(* Schneider Machine Expert - Basic project Tarea1C3_TomasMoreno, file version 2.7.0.0 *)
(* ProjectInformations: Name=Nuevo proyecto *)

HARDWARE
  Cpu 0: TM221CE16R
  EthernetConfiguration: NetworkName=M221, IpAllocationMode=FixedAddress, IpAddress=0.0.0.0, SubnetMask=0.0.0.0
  SerialLineConfiguration: Baud=Baud19200, Parity=ParityEven, DataBits=DataBits8, StopBits=StopBits1, PhysicalMedium=PhysicalMediumRs485, TransmissionMode=TransmissionModeModbusRtu, SlaveId=1, Addressing=SlaveAddressing
  MastTask: UsePeriodScanMode=false, PeriodScan=100
  FastTask: Period=255
  CpuBehavior: StartingMode=StartAsPreviousState, AutoSaveRamOnEeprom=true, WatchdogPeriod=250

SYMBOLS  (address, symbol, comment, settings)
  %M0         "PARTIR"
  %M1         "PARAR"
  %M2         "AUTOMATICO"
  %M3         "MANUAL"
  %M4         "RESETEO"
  %M5         "PARADA DE EMERGENCIA"
  %M6         "SENSOR TRANSPORTE"
  %M7         "SENSOR CONTADOR CP"
  %M8         "SENSOR CONTADOR CG"
  %M9         "IMPULSADOR CAJAS (MANUAL)"
  %M20        "LED PARTIR"
  %M21        "LED RESET"
  %M22        "LED PARAR"
  %M23        "LED FUNCIONAMIENTO SISTEMA"
  %M24        "LED CONTADOR CP"
  %M25        "LED CONTADOR CG"
  %M26        "CORREA PRINCIPAL"
  %M27        "TRANSPORTE ADELANTE"
  %M28        "TRANSPORTE CG"
  %M29        "TRANSPORTE CP"
  %M30        "CORREA CAJAS GRANDES"
  %M31        "CORREA CAJAS PEQUEÑAS"
  %M32        "EMISOR DE CAJAS"
  %M33        "LED IMPULSADOR MANUAL"
  %M50        "ARRANQUE SISTEMA"
  %M61        "S_TRANSP_CG"
  %M62        "S_TRANSP_CP"
  %M63        "H_TRANSP_CG"
  %M64        "H_TRANSP_CP"
  %S6       SB_TB1S  "Base de tiempo de 1 s generada por un reloj interno"
  %TM0        [Type=TOF, Preset=1, Base=OneSecond]
  %TM1        [Type=TOF, Preset=1, Base=OneSecond]
  %C0         [Preset=1]
  %C1         [Preset=1]

POU Nuevo POU
  (* SectionNumber=1 *)

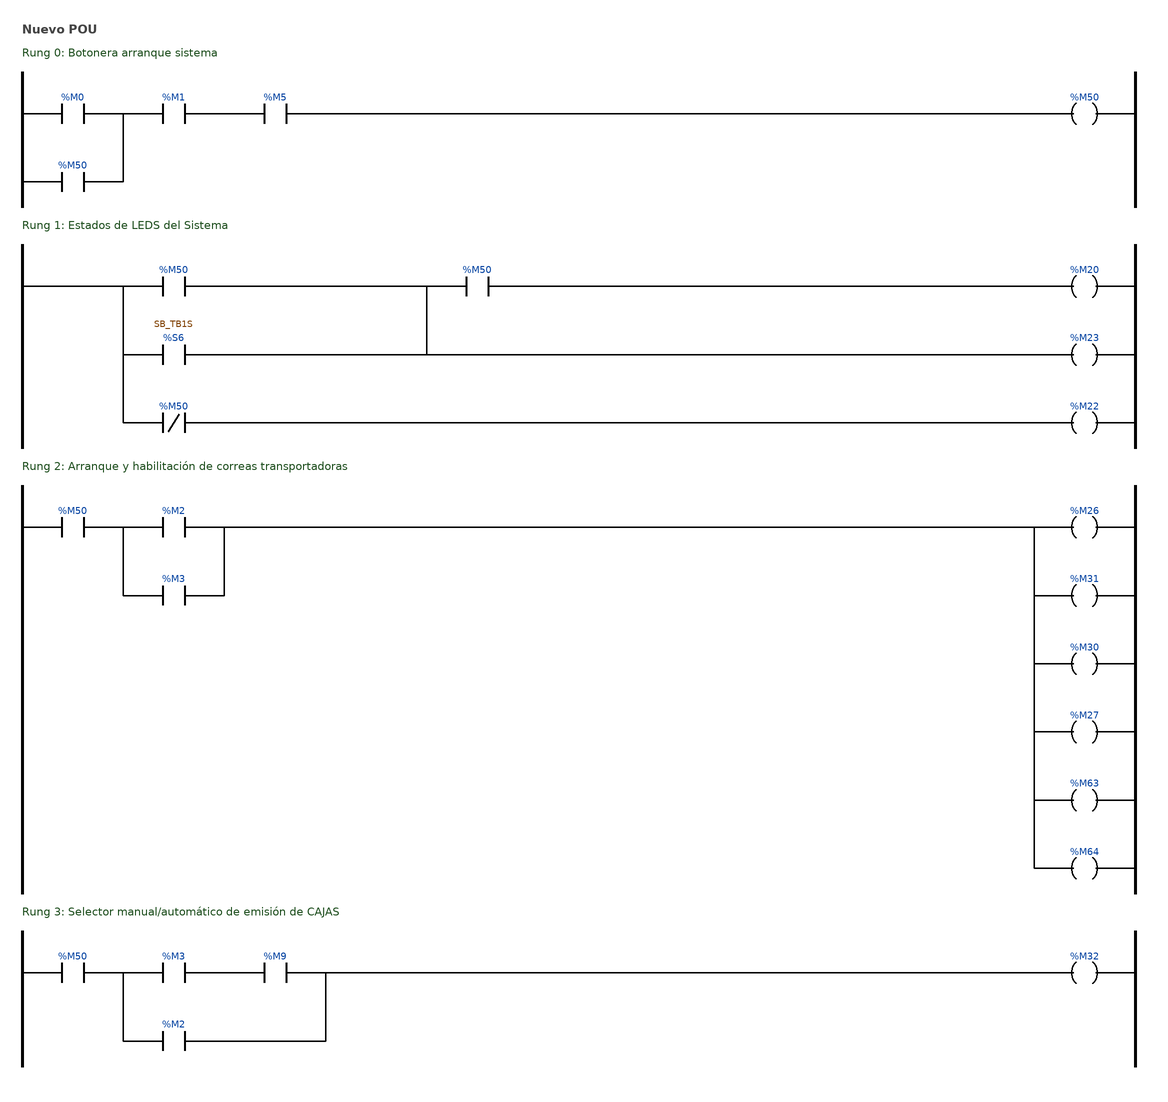

// Rung 0: Botonera arranque sistema
  LD %M0
  OR %M50
  AND %M1
  AND %M5
  ST %M50
  // as ST:
  //   %M50 := (%M0 OR %M50) AND %M1 AND %M5;

// Rung 1: Estados de LEDS del Sistema
  LD 1
  MPS
  AND( %M50
  OR %S6                  (* SB_TB1S *)
  )
  MPS
  AND %M50
  ST %M20
  MPP
  ST %M23
  MPP
  ANDN %M50
  ST %M22
  // as ST:
  //   %M20 := (%M50 OR SB_TB1S) AND %M50;
  //   %M23 := %M50 OR SB_TB1S;
  //   %M22 := NOT %M50;

// Rung 2: Arranque y habilitación de correas transportadoras
  LD %M50
  AND( %M2
  OR %M3
  )
  ST %M26
  ST %M31
  ST %M30
  ST %M27
  ST %M63
  ST %M64
  // as ST:
  //   %M26 := %M50 AND (%M2 OR %M3);
  //   %M31 := %M50 AND (%M2 OR %M3);
  //   %M30 := %M50 AND (%M2 OR %M3);
  //   %M27 := %M50 AND (%M2 OR %M3);
  //   %M63 := %M50 AND (%M2 OR %M3);
  //   %M64 := %M50 AND (%M2 OR %M3);

// Rung 3: Selector manual/automático de emisión de CAJAS
  LD %M50
  AND( %M3
  AND %M9
  OR %M2
  )
  ST %M32
  // as ST:
  //   %M32 := %M50 AND (%M3 AND %M9 OR %M2);

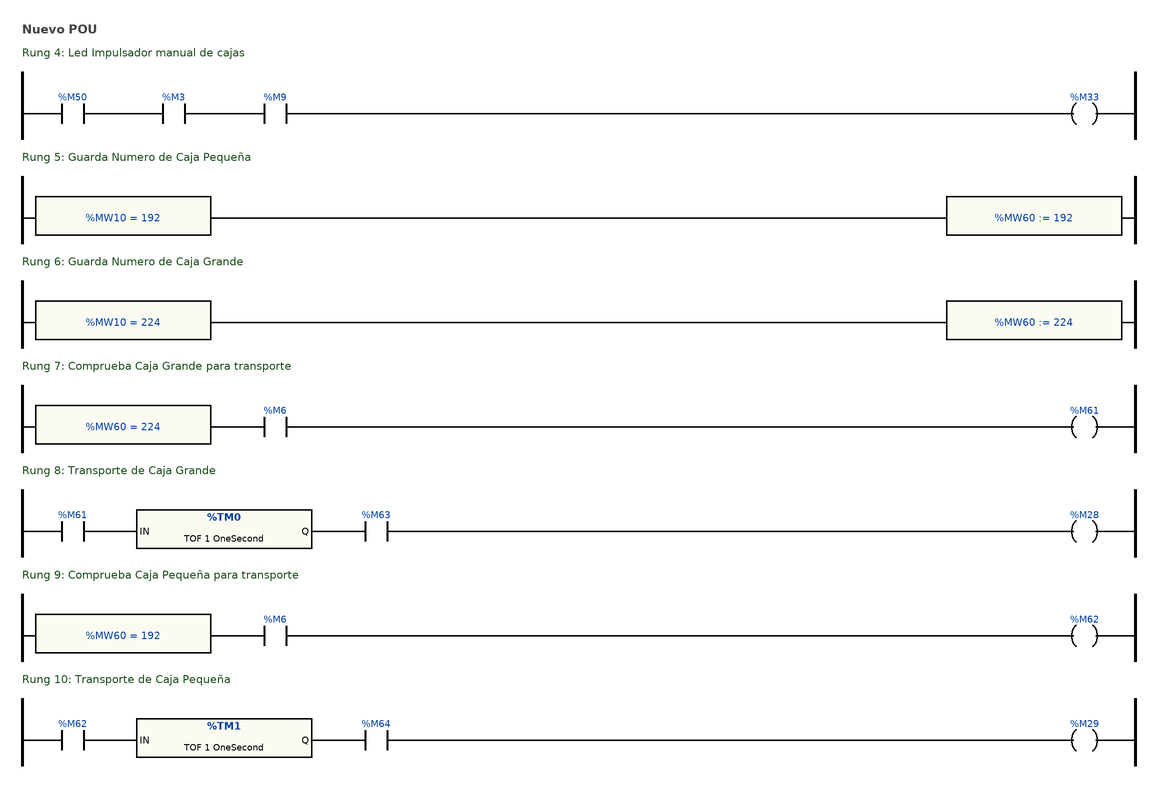

// Rung 4: Led Impulsador manual de cajas
  LD %M50
  AND %M3
  AND %M9
  ST %M33
  // as ST:
  //   %M33 := %M50 AND %M3 AND %M9;

// Rung 5: Guarda Numero de Caja Pequeña
  LD [ %MW10 = 192 ]
  [ %MW60 := 192 ]
  // as ST:
  //   IF %MW10 = 192 THEN %MW60 := 192; END_IF;

// Rung 6: Guarda Numero de Caja Grande
  LD [ %MW10 = 224 ]
  [ %MW60 := 224 ]
  // as ST:
  //   IF %MW10 = 224 THEN %MW60 := 224; END_IF;

// Rung 7: Comprueba Caja Grande para transporte
  LD [ %MW60 = 224 ]
  AND %M6
  ST %M61
  // as ST:
  //   %M61 := %MW60 = 224 AND %M6;

// Rung 8: Transporte de Caja Grande
  BLK %TM0
  LD %M61
  IN
  OUT_BLK
  LD Q
  AND %M63
  ST %M28
  END_BLK
  // as ST:
  //   %TM0(IN := %M61);
  //   %M28 := %TM0.Q AND %M63;

// Rung 9: Comprueba Caja Pequeña para transporte
  LD [ %MW60 = 192 ]
  AND %M6
  ST %M62
  // as ST:
  //   %M62 := %MW60 = 192 AND %M6;

// Rung 10: Transporte de Caja Pequeña
  BLK %TM1
  LD %M62
  IN
  OUT_BLK
  LD Q
  AND %M64
  ST %M29
  END_BLK
  // as ST:
  //   %TM1(IN := %M62);
  //   %M29 := %TM1.Q AND %M64;

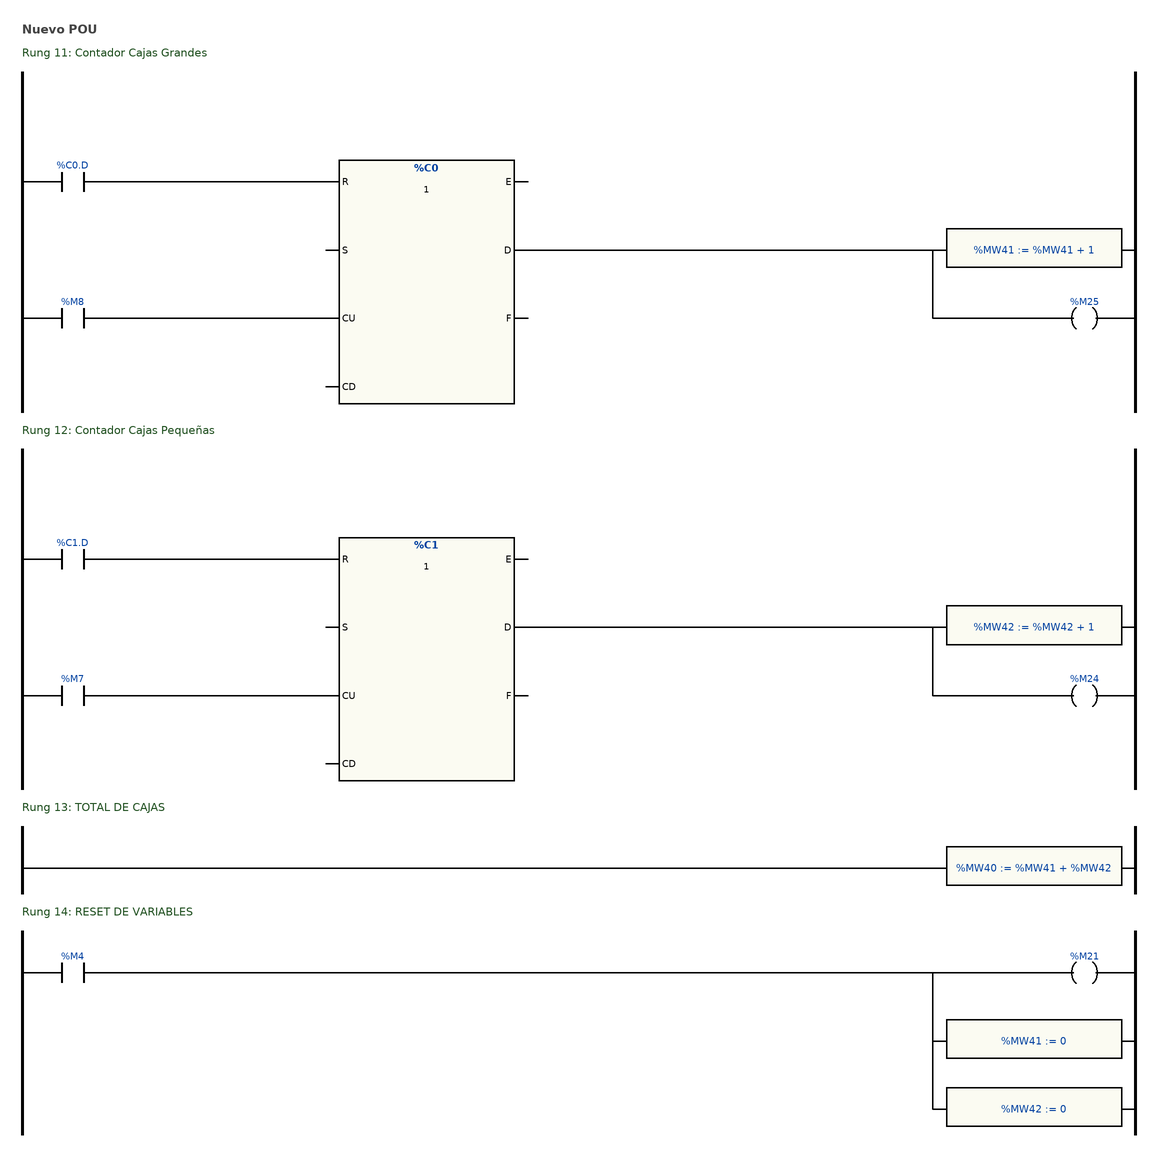

// Rung 11: Contador Cajas Grandes
  BLK %C0
  LD %C0.D
  R
  LD %M8
  CU
  OUT_BLK
  LD D
  [ %MW41 := %MW41 + 1 ]
  ST %M25
  END_BLK
  // as ST:
  //   %C0(R := %C0.D, CU := %M8);
  //   IF %C0.D THEN %MW41 := %MW41 + 1; END_IF;
  //   %M25 := %C0.D;

// Rung 12: Contador Cajas Pequeñas
  BLK %C1
  LD %C1.D
  R
  LD %M7
  CU
  OUT_BLK
  LD D
  [ %MW42 := %MW42 + 1 ]
  ST %M24
  END_BLK
  // as ST:
  //   %C1(R := %C1.D, CU := %M7);
  //   IF %C1.D THEN %MW42 := %MW42 + 1; END_IF;
  //   %M24 := %C1.D;

// Rung 13: TOTAL DE CAJAS
  LD 1
  [ %MW40 := %MW41 + %MW42 ]
  // as ST:
  //   %MW40 := %MW41 + %MW42;

// Rung 14: RESET DE VARIABLES
  LD %M4
  ST %M21
  [ %MW41 := 0 ]
  [ %MW42 := 0 ]
  // as ST:
  //   %M21 := %M4;
  //   IF %M4 THEN %MW41 := 0; END_IF;
  //   IF %M4 THEN %MW42 := 0; END_IF;
